INTERFACE I_EPSSamplePaddleGasNeedle


METHOD CheckAndActivateIfRequired
VAR_IN_OUT
	StageZSamplePaddle	: lcls_twincat_motion.ST_MotionStage;
	StageZGasNeedle	: lcls_twincat_motion.ST_MotionStage;
END_VAR
END_METHOD

END_INTERFACE

(* stored: Version 1.1.0.1, ProductVersion 3.1.4022.18
   Itf I_EPSSamplePaddleGasNeedle: Id {debb4a44-0f7b-4d07-a00c-44fef871f029}
   Method CheckAndActivateIfRequired: Id {d5099148-0ad2-4c97-a699-5b94edabef05} *)
